INTERFACE ITcoCustomizedDialogAnswer EXTENDS ITcoCustomizedDialogFormat

PROPERTY Answer : ecustomizedDialogAnswer
GET
END_GET
END_PROPERTY

END_INTERFACE

(* stored: Version 1.1.0.1
   Itf ITcoCustomizedDialogAnswer: Id {114446a6-3bf5-02e2-334f-93684d65d8dc}
   Property Answer: Id {a337f277-b9f4-0ef3-1e12-deaebf20924a}
   Get Get: Id {a6757865-7a3a-03d8-0a1a-91dadcb685cc} *)
